KUKA KRL data list: ps_b_etb_res_c02.dat

&ACCESS RVO1
&COMMENT Solda Atego ETB
DEFDAT ps_b_etb_res_c02
;FOLD EXTERNAL DECLARATIONS;%{PE}%V2.2.2,%MKUKATPBASIS,%CEXT,%VCOMMON,%P
;FOLD BAS EXT;%{PE}%V2.2.2,%MKUKATPBASIS,%CEXT,%VEXT,%P
EXT  BAS (BAS_COMMAND  :IN,REAL  :IN )
DECL INT SUCCESS
;ENDFOLD
;FOLD A10 EXT;%{E}%V2.2.2,%MKUKATPARC,%CEXT,%VEXT,%P
EXT  A10 (A_CMD_T  :IN,A_STRT_T  :IN,A_WELD_T  :IN,A_END_T  :IN,INT  :IN )
;ENDFOLD
;FOLD A20 EXT;%{E}%V2.2.2,%MKUKATPA20,%CEXT,%VEXT,%P
EXT  A20 (INT  :IN,WELD_ST  :IN,WELD_FI  :IN,INT  :IN )
;ENDFOLD
;FOLD GRIPPER EXT;%{E}%V2.2.2,%MKUKATPGRIPPER,%CEXT,%VEXT,%P
EXT  H50 (INT  :IN,INT  :IN,INT  :IN,GRP_TYP  :IN )
;ENDFOLD
;FOLD SPOT EXT;%{E}%V2.2.2,%MKUKATPSPOT,%CEXT,%VEXT,%P
EXT  USERSPOT (S_COMMAND  :IN,SPOT_TYPE  :IN )
;ENDFOLD
;FOLD TOUCHSENSE EXT;%{E}%V2.2.2,%MKUKATPTS,%CEXT,%VEXT,%P
EXT  H70 (INT  :IN,SRCH_TYP_2  :OUT,E6POS  :IN,SRCH_TYP_3  :IN,SRCH_TYP_2  :IN,SRCH_TYP_2  :IN,SRCH_TYP_2  :IN,SRCH_TYP_2  :IN,SRCH_TYP_2  :IN,INT  :IN )
;ENDFOLD
;FOLD USER EXT;%{}%V2.2.2,%MKUKATPUSER,%CEXT,%VEXT,%P
;Make here your modifications
;ENDFOLD
;ENDFOLD

DECL FDAT Fl005={TOOL_NO 3,BASE_NO 3,IPO_FRAME #BASE}
DECL PDAT PP_OLP2={VEL 100.0,ACC 100.0,APO_DIST 0.0}
DECL E6POS Xl005={x -259.953003,y 860.291992,z 674.213013,a 106.465103,b 65.7322998,c -50.9701004,s 2,t 42}
DECL FDAT Fl010={TOOL_NO 3,BASE_NO 3,IPO_FRAME #BASE}
DECL PDAT PP_OLP3={VEL 100.0,ACC 100.0,APO_DIST 0.0}
DECL E6POS Xl010={x 238.578995,y 878.294983,z 634.81897,a 106.465103,b 65.7322998,c -50.9701004,s 2,t 43}
DECL FDAT Fl015={TOOL_NO 3,BASE_NO 3,IPO_FRAME #BASE}
DECL PDAT PP_OLP4={VEL 100.0,ACC 100.0,APO_DIST 0.0}
DECL E6POS Xl015={x 233.995102,y 927.062683,z 508.398987,a 106.4627,b 65.7314301,c -48.9741592,s 2,t 43,e1 0.0,e2 0.0,e3 0.0,e4 0.0,e5 0.0,e6 0.0}
DECL LDAT LL_OLP1={VEL 2.0,ACC 100.0,APO_DIST 0.0,APO_FAC 0.0}
DECL FDAT Fl020={TOOL_NO 3,BASE_NO 3,IPO_FRAME #BASE}
DECL PDAT PP_OLP5={VEL 100.0,ACC 100.0,APO_DIST 0.0}
DECL E6POS Xl020={x 240.050705,y 924.635925,z 506.612305,a 106.462997,b 65.7332382,c -48.9725304,s 2,t 43,e1 0.0,e2 0.0,e3 0.0,e4 0.0,e5 0.0,e6 0.0}
DECL FDAT Fl025={TOOL_NO 3,BASE_NO 3,IPO_FRAME #BASE}
DECL PDAT PP_OLP6={VEL 100.0,ACC 100.0,APO_DIST 0.0}
DECL E6POS Xl025={x 230.037399,y 926.909119,z 610.785889,a 106.4646,b 65.7323837,c -48.9705811,s 2,t 43,e1 0.0,e2 0.0,e3 0.0,e4 0.0,e5 0.0,e6 0.0}
DECL FDAT Fl030={TOOL_NO 3,BASE_NO 3,IPO_FRAME #BASE}
DECL PDAT PP_OLP7={VEL 100.0,ACC 100.0,APO_DIST 0.0}
DECL E6POS Xl030={x 193.569397,y 878.43573,z 618.731201,a 136.368896,b 76.3886337,c -42.6437798,s 2,t 43,e1 0.0,e2 0.0,e3 0.0,e4 0.0,e5 0.0,e6 0.0}
DECL E6POS Xl011={x 216.297104,y 817.987915,z 621.025818,a -90.0010071,b 86.8945236,c 89.9989166,s 2,t 43,e1 0.0,e2 0.0,e3 0.0,e4 0.0,e5 0.0,e6 0.0}
DECL FDAT Fl011={TOOL_NO 3,BASE_NO 3,IPO_FRAME #BASE}
DECL PDAT PP_OLP11={VEL 100.0,ACC 100.0,APO_DIST 0.0}
DECL E6POS Xl016={x 211.330002,y 837.989685,z 424.030212,a -89.9980164,b 86.8946533,c 90.0018005,s 2,t 43,e1 0.0,e2 0.0,e3 0.0,e4 0.0,e5 0.0,e6 0.0}
DECL FDAT Fl016={TOOL_NO 3,BASE_NO 3,IPO_FRAME #BASE}
DECL PDAT PP_OLP12={VEL 100.0,ACC 100.0,APO_DIST 0.0}
DECL E6POS XSWP_60_7354={x 203.809906,y 837.713989,z 419.105103,a -90.024231,b 86.8921432,c 89.974617,s 2,t 43,e1 0.0,e2 0.0,e3 0.0,e4 0.0,e5 0.0,e6 0.0}
DECL FDAT FSWP_60_7354={TOOL_NO 3,BASE_NO 3,IPO_FRAME #BASE}
DECL LDAT LL_OLP2={VEL 2.0,ACC 100.0,APO_DIST 0.0,APO_FAC 0.0}
DECL E6POS XSWP_60_7356={x 204.900299,y 813.062012,z 427.303589,a -90.0252304,b 86.8959122,c 89.9749298,s 2,t 43,e1 0.0,e2 0.0,e3 0.0,e4 0.0,e5 0.0,e6 0.0}
DECL FDAT FSWP_60_7356={TOOL_NO 3,BASE_NO 3,IPO_FRAME #BASE}
DECL LDAT LL_OLP3={VEL 2.0,ACC 100.0,APO_DIST 0.0,APO_FAC 0.0}
DECL E6POS XSWP_60_7358={x 205.666595,y 785.228699,z 444.857788,a -90.0419312,b 86.8953781,c 89.9582901,s 2,t 43,e1 0.0,e2 0.0,e3 0.0,e4 0.0,e5 0.0,e6 0.0}
DECL FDAT FSWP_60_7358={TOOL_NO 3,BASE_NO 3,IPO_FRAME #BASE}
DECL LDAT LL_OLP4={VEL 2.0,ACC 100.0,APO_DIST 0.0,APO_FAC 0.0}
DECL E6POS XSWP_60_7360={x 203.261703,y 756.455627,z 466.485809,a -89.9985809,b 86.8937683,c 90.0012436,s 2,t 43,e1 0.0,e2 0.0,e3 0.0,e4 0.0,e5 0.0,e6 0.0}
DECL FDAT FSWP_60_7360={TOOL_NO 3,BASE_NO 3,IPO_FRAME #BASE}
DECL LDAT LL_OLP5={VEL 2.0,ACC 100.0,APO_DIST 0.0,APO_FAC 0.0}
DECL E6POS XSWP_60_7362={x 206.944794,y 725.337585,z 475.673492,a 89.9988937,b 70.9206924,c -90.0019226,s 2,t 43,e1 0.0,e2 0.0,e3 0.0,e4 0.0,e5 0.0,e6 0.0}
DECL FDAT FSWP_60_7362={TOOL_NO 3,BASE_NO 3,IPO_FRAME #BASE}
DECL LDAT LL_OLP6={VEL 2.0,ACC 100.0,APO_DIST 0.0,APO_FAC 0.0}
DECL E6POS XSWP_60_7364={x 206.622696,y 692.928894,z 476.588287,a -90.0024414,b 86.1575623,c 89.9975586,s 2,t 43,e1 0.0,e2 0.0,e3 0.0,e4 0.0,e5 0.0,e6 0.0}
DECL FDAT FSWP_60_7364={TOOL_NO 3,BASE_NO 3,IPO_FRAME #BASE}
DECL LDAT LL_OLP7={VEL 2.0,ACC 100.0,APO_DIST 0.0,APO_FAC 0.0}
DECL E6POS XSWP_60_7366={x 203.315002,y 660.348389,z 476.359894,a -90.0006638,b 56.1120415,c 89.9992981,s 2,t 43,e1 0.0,e2 0.0,e3 0.0,e4 0.0,e5 0.0,e6 0.0}
DECL FDAT FSWP_60_7366={TOOL_NO 3,BASE_NO 3,IPO_FRAME #BASE}
DECL LDAT LL_OLP8={VEL 2.0,ACC 100.0,APO_DIST 0.0,APO_FAC 0.0}
DECL E6POS XSWP_60_7368={x 206.116501,y 634.32843,z 476.098907,a -90.0014801,b 58.2454681,c 90.0003967,s 2,t 43,e1 0.0,e2 0.0,e3 0.0,e4 0.0,e5 0.0,e6 0.0}
DECL FDAT FSWP_60_7368={TOOL_NO 3,BASE_NO 3,IPO_FRAME #BASE}
DECL LDAT LL_OLP9={VEL 2.0,ACC 100.0,APO_DIST 0.0,APO_FAC 0.0}
DECL E6POS XSWP_60_7370={x 205.649307,y 608.364075,z 476.227295,a -90.000618,b 59.0425911,c 89.9998627,s 2,t 43,e1 0.0,e2 0.0,e3 0.0,e4 0.0,e5 0.0,e6 0.0}
DECL FDAT FSWP_60_7370={TOOL_NO 3,BASE_NO 3,IPO_FRAME #BASE}
DECL LDAT LL_OLP10={VEL 2.0,ACC 100.0,APO_DIST 0.0,APO_FAC 0.0}
DECL E6POS XSWP_60_7372={x 207.227097,y 582.377502,z 476.378601,a -90.0000229,b 59.7199898,c 90.0000229,s 2,t 43,e1 0.0,e2 0.0,e3 0.0,e4 0.0,e5 0.0,e6 0.0}
DECL FDAT FSWP_60_7372={TOOL_NO 3,BASE_NO 3,IPO_FRAME #BASE}
DECL LDAT LL_OLP11={VEL 2.0,ACC 100.0,APO_DIST 0.0,APO_FAC 0.0}
DECL E6POS XSWP_60_7374={x 206.739594,y 556.385376,z 476.24881,a -89.9996872,b 60.0724792,c 89.9999695,s 2,t 43,e1 0.0,e2 0.0,e3 0.0,e4 0.0,e5 0.0,e6 0.0}
DECL FDAT FSWP_60_7374={TOOL_NO 3,BASE_NO 3,IPO_FRAME #BASE}
DECL LDAT LL_OLP12={VEL 2.0,ACC 100.0,APO_DIST 0.0,APO_FAC 0.0}
DECL E6POS Xl026={x 232.763107,y 556.379089,z 476.253387,a -89.9998627,b 59.855629,c 90.0001068,s 2,t 43,e1 0.0,e2 0.0,e3 0.0,e4 0.0,e5 0.0,e6 0.0}
DECL FDAT Fl026={TOOL_NO 3,BASE_NO 3,IPO_FRAME #BASE}
DECL PDAT PP_OLP14={VEL 100.0,ACC 100.0,APO_DIST 0.0}
DECL E6POS Xl031={x 237.137695,y 429.935913,z 476.3927,a -90.001503,b 59.8552017,c 89.9993286,s 2,t 43,e1 0.0,e2 0.0,e3 0.0,e4 0.0,e5 0.0,e6 0.0}
DECL FDAT Fl031={TOOL_NO 3,BASE_NO 3,IPO_FRAME #BASE}
DECL PDAT PP_OLP15={VEL 100.0,ACC 100.0,APO_DIST 0.0}
DECL E6POS XSWP_60_7376={x 205.848206,y 441.043304,z 482.712006,a -89.9979706,b 60.0047493,c 90.0008774,s 2,t 43,e1 0.0,e2 0.0,e3 0.0,e4 0.0,e5 0.0,e6 0.0}
DECL FDAT FSWP_60_7376={TOOL_NO 3,BASE_NO 3,IPO_FRAME #BASE}
DECL LDAT LL_OLP13={VEL 2.0,ACC 100.0,APO_DIST 0.0,APO_FAC 0.0}
DECL E6POS XSWP_60_7378={x 206.973907,y 431.014099,z 441.041809,a -89.9991226,b 61.5301018,c 90.0008698,s 2,t 43,e1 0.0,e2 0.0,e3 0.0,e4 0.0,e5 0.0,e6 0.0}
DECL FDAT FSWP_60_7378={TOOL_NO 3,BASE_NO 3,IPO_FRAME #BASE}
DECL LDAT LL_OLP14={VEL 2.0,ACC 100.0,APO_DIST 0.0,APO_FAC 0.0}
DECL E6POS XSWP_60_7380={x 206.840393,y 416.639099,z 400.304108,a -89.9998703,b 62.6937904,c 90.0006027,s 2,t 43,e1 0.0,e2 0.0,e3 0.0,e4 0.0,e5 0.0,e6 0.0}
DECL FDAT FSWP_60_7380={TOOL_NO 3,BASE_NO 3,IPO_FRAME #BASE}
DECL LDAT LL_OLP15={VEL 2.0,ACC 100.0,APO_DIST 0.0,APO_FAC 0.0}
DECL E6POS XSWP_60_7220={x 205.599396,y 39.2980804,z 386.423615,a -89.9959183,b 44.4748917,c 89.9934921,s 2,t 43,e1 0.0,e2 0.0,e3 0.0,e4 0.0,e5 0.0,e6 0.0}
DECL FDAT FSWP_60_7220={TOOL_NO 3,BASE_NO 3,IPO_FRAME #BASE}
DECL E6POS XSWP_60_7222={x 206.282593,y 88.0883484,z 386.359711,a -89.9976273,b 44.4760399,c 89.9922333,s 2,t 43,e1 0.0,e2 0.0,e3 0.0,e4 0.0,e5 0.0,e6 0.0}
DECL FDAT FSWP_60_7222={TOOL_NO 3,BASE_NO 3,IPO_FRAME #BASE}
DECL LDAT LL_OLP31={VEL 2.0,ACC 50.0,APO_DIST 0.0,APO_FAC 0.0}
DECL LDAT LL_OLP32={VEL 2.0,ACC 50.0,APO_DIST 0.0,APO_FAC 0.0}
DECL LDAT LL_OLP33={VEL 2.0,ACC 100.0,APO_DIST 0.0,APO_FAC 0.0}
DECL LDAT LL_OLP34={VEL 2.0,ACC 100.0,APO_DIST 0.0,APO_FAC 0.0}
DECL E6POS XSWP_60_7260={x 181.102097,y 50.2497406,z 492.070099,a -80.3131027,b 32.1295509,c 107.793098,s 2,t 11,e1 0.0,e2 0.0,e3 0.0,e4 0.0,e5 0.0,e6 0.0}
DECL FDAT FSWP_60_7260={TOOL_NO 3,BASE_NO 3,IPO_FRAME #BASE}
DECL E6POS XSWP_60_7261={x 180.671097,y 1.26443899,z 490.916901,a -80.5087128,b 31.6135597,c 107.6959,s 2,t 11,e1 0.0,e2 0.0,e3 0.0,e4 0.0,e5 0.0,e6 0.0}
DECL FDAT FSWP_60_7261={TOOL_NO 3,BASE_NO 3,IPO_FRAME #BASE}
DECL LDAT LL_OLP36={VEL 2.0,ACC 100.0,APO_DIST 0.0,APO_FAC 0.0}
DECL LDAT LL_OLP37={VEL 2.0,ACC 100.0,APO_DIST 0.0,APO_FAC 0.0}
DECL LDAT LL_OLP38={VEL 2.0,ACC 100.0,APO_DIST 0.0,APO_FAC 0.0}
DECL E6POS Xl086={x 160.914307,y 87.6342468,z 584.528687,a -71.1530838,b 50.3254509,c 113.916496,s 2,t 43,e1 0.0,e2 0.0,e3 0.0,e4 0.0,e5 0.0,e6 0.0}
DECL FDAT Fl086={TOOL_NO 3,BASE_NO 3,IPO_FRAME #BASE}
DECL PDAT PP_OLP49={VEL 100.0,ACC 100.0,APO_DIST 0.0}
DECL E6POS Xl091={x 172.296906,y 391.390808,z 683.738708,a -90.0011826,b 46.4089699,c 90.0007324,s 2,t 43,e1 0.0,e2 0.0,e3 0.0,e4 0.0,e5 0.0,e6 0.0}
DECL FDAT Fl091={TOOL_NO 3,BASE_NO 3,IPO_FRAME #BASE}
DECL PDAT PP_OLP50={VEL 100.0,ACC 100.0,APO_DIST 0.0}
DECL E6POS Xl096={x -352.044708,y 791.362305,z 674.194885,a 102.528297,b 65.7295227,c -50.9826317,s 2,t 42,e1 0.0,e2 0.0,e3 0.0,e4 0.0,e5 0.0,e6 0.0}
DECL FDAT Fl096={TOOL_NO 3,BASE_NO 3,IPO_FRAME #BASE}
DECL PDAT PP_OLP51={VEL 100.0,ACC 100.0,APO_DIST 0.0}
DECL E6POS XSWP_60_9320={x 233.906906,y 930.794983,z 509.773987,a 106.517899,b 65.7420273,c -48.8959618,s 2,t 43,e1 0.0,e2 0.0,e3 0.0,e4 0.0,e5 0.0,e6 0.0}
DECL FDAT FSWP_60_9320={TOOL_NO 3,BASE_NO 3,IPO_FRAME #BASE}
DECL E6POS XP6={x -1383.52795,y 1084.21204,z 300.229401,a 152.116806,b 8.17701721,c 8.23256302,s 2,t 42,e1 0.0,e2 0.0,e3 0.0,e4 0.0,e5 0.0,e6 0.0}
DECL FDAT FP6={TOOL_NO 3,BASE_NO 3,IPO_FRAME #BASE}
DECL PDAT PPDAT6={VEL 100.0,ACC 100.0,APO_DIST 0.0}
DECL E6POS XP7={x 211.5793,y 905.759277,z 610.608276,a 118.261002,b 68.8623581,c -44.6343498,s 2,t 43,e1 0.0,e2 0.0,e3 0.0,e4 0.0,e5 0.0,e6 0.0}
DECL FDAT FP7={TOOL_NO 3,BASE_NO 3,IPO_FRAME #BASE}
DECL PDAT PPDAT7={VEL 100.0,ACC 100.0,APO_DIST 0.0}
DECL SPOT_SUGG_T LAST_SPOT={GUN[] "3                       ",RETR_CMD[] "#OPN                    ",CHOISE[] "#FIRST                  ",CLO_TM[] "1                       ",PGNO1[] "197                     ",PRESS1[] "0                       ",PGNO2[] "1                       ",PRESS2[] "0                       ",SPOT_PARAMS[] "NORMAL                  "}
DECL BASIS_SUGG_T LAST_BASIS={POINT1[] "SWP_60_9234             ",POINT2[] "SWP_60_9234             ",CP_PARAMS[] "CPDAT30                 ",PTP_PARAMS[] "PDAT38                  ",CONT[] "                        ",CP_VEL[] "2                       ",PTP_VEL[] "100                     "}
DECL E6POS XSWP_60_7258={x 177.344299,y 91.2774734,z 492.510498,a -80.9878082,b 30.2983799,c 107.447899,s 2,t 11,e1 0.0,e2 0.0,e3 0.0,e4 0.0,e5 0.0,e6 0.0}
DECL FDAT FSWP_60_7258={TOOL_NO 3,BASE_NO 3,IPO_FRAME #BASE}
DECL E6POS XSWP_60_7217={x 212.0215,y -5.72816896,z 386.457611,a -89.9976273,b 44.4766617,c 89.9928436,s 2,t 43,e1 0.0,e2 0.0,e3 0.0,e4 0.0,e5 0.0,e6 0.0}
DECL FDAT FSWP_60_7217={TOOL_NO 3,BASE_NO 3,IPO_FRAME #BASE}
DECL E6POS XSWP_60_7218={x 230.446198,y 232.953796,z 499.446594,a -89.995369,b 44.4764595,c 89.9949036,s 2,t 43,e1 0.0,e2 0.0,e3 0.0,e4 0.0,e5 0.0,e6 0.0}
DECL FDAT FSWP_60_7218={TOOL_NO 3,BASE_NO 3,IPO_FRAME #BASE}
DECL PDAT PPDAT1={VEL 100.0,ACC 100.0,APO_DIST 0.0}
DECL E6POS XSWP_60_7253={x 183.271103,y -168.511398,z 488.607788,a -80.492569,b 31.5890808,c 107.705902,s 2,t 43,e1 0.0,e2 0.0,e3 0.0,e4 0.0,e5 0.0,e6 0.0}
DECL FDAT FSWP_60_7253={TOOL_NO 3,BASE_NO 3,IPO_FRAME #BASE}
DECL E6POS XSWP_60_7255={x 182.816605,y -136.932495,z 488.353302,a -80.4999466,b 31.6015491,c 107.701401,s 2,t 43,e1 0.0,e2 0.0,e3 0.0,e4 0.0,e5 0.0,e6 0.0}
DECL FDAT FSWP_60_7255={TOOL_NO 3,BASE_NO 3,IPO_FRAME #BASE}
DECL E6POS XSWP_60_7257={x 182.301605,y -88.3556519,z 488.131897,a -80.5033569,b 31.6069908,c 107.6978,s 2,t 43,e1 0.0,e2 0.0,e3 0.0,e4 0.0,e5 0.0,e6 0.0}
DECL FDAT FSWP_60_7257={TOOL_NO 3,BASE_NO 3,IPO_FRAME #BASE}
DECL E6POS XSWP_60_7262={x 180.669205,y 1.25821102,z 490.930298,a -80.508873,b 31.6130199,c 107.696198,s 2,t 11,e1 0.0,e2 0.0,e3 0.0,e4 0.0,e5 0.0,e6 0.0}
DECL FDAT FSWP_60_7262={TOOL_NO 3,BASE_NO 3,IPO_FRAME #BASE}
DECL SPOT_TYPE SNORMAL
DECL SPOT_TYPE SNORMAL28
DECL E6POS XP15={x -800.207581,y 1052.86096,z 371.426514,a 42.3493195,b -1.00002205,c -26.3774109,s 2,t 42,e1 0.0,e2 0.0,e3 0.0,e4 0.0,e5 0.0,e6 0.0}
DECL FDAT FP15={TOOL_NO 1,BASE_NO 3,IPO_FRAME #BASE}
DECL PDAT PPDAT2={VEL 100.0,ACC 100.0,APO_DIST 100.0}
DECL E6POS Xl048={x 235.096298,y 205.879898,z 399.392609,a -89.9929504,b 44.4753685,c 89.9981766,s 2,t 43,e1 0.0,e2 0.0,e3 0.0,e4 0.0,e5 0.0,e6 0.0}
DECL FDAT Fl048={TOOL_NO 3,BASE_NO 3,IPO_FRAME #BASE}
DECL PDAT PP_OLP53={VEL 100.0,ACC 100.0,APO_DIST 0.0}
DECL LDAT LL_OLP50={VEL 2.0,ACC 100.0,APO_DIST 0.0,APO_FAC 0.0}
DECL SPOT_TYPE SNORMAL29
DECL LDAT LCPDAT5={VEL 2.0,ACC 100.0,APO_DIST 100.0,APO_FAC 50.0}
DECL LDAT LCPDAT6={VEL 2.0,ACC 100.0,APO_DIST 100.0,APO_FAC 50.0}
DECL E6POS XP16={x 208.831604,y -34.5271187,z 495.562012,a -80.5012817,b 31.5980301,c 107.702202,s 2,t 11,e1 0.0,e2 0.0,e3 0.0,e4 0.0,e5 0.0,e6 0.0}
DECL FDAT FP16={TOOL_NO 3,BASE_NO 3,IPO_FRAME #BASE}
DECL LDAT LCPDAT7={VEL 2.0,ACC 50.0,APO_DIST 100.0,APO_FAC 50.0}
DECL E6POS XSWP_60_7381={x 206.840393,y 416.639099,z 400.304108,a -89.9998703,b 62.6937904,c 90.0006027,s 2,t 43,e1 0.0,e2 0.0,e3 0.0,e4 0.0,e5 0.0,e6 0.0}
DECL FDAT FSWP_60_7381={TOOL_NO 3,BASE_NO 3,IPO_FRAME #BASE}
DECL LDAT LL_OLP16={VEL 2.0,ACC 100.0,APO_DIST 0.0,APO_FAC 0.0}
DECL SPOT_TYPE SNORMAL13
DECL E6POS XSWP_60_7382={x 206.840393,y 416.639099,z 400.304108,a -89.9998703,b 62.6937904,c 90.0006027,s 2,t 43,e1 0.0,e2 0.0,e3 0.0,e4 0.0,e5 0.0,e6 0.0}
DECL FDAT FSWP_60_7382={TOOL_NO 3,BASE_NO 3,IPO_FRAME #BASE}
DECL LDAT LL_OLP17={VEL 2.0,ACC 100.0,APO_DIST 0.0,APO_FAC 0.0}
DECL E6POS XSWP_60_7383={x 206.840393,y 416.639099,z 400.304108,a -89.9998703,b 62.6937904,c 90.0006027,s 2,t 43,e1 0.0,e2 0.0,e3 0.0,e4 0.0,e5 0.0,e6 0.0}
DECL FDAT FSWP_60_7383={TOOL_NO 3,BASE_NO 3,IPO_FRAME #BASE}
DECL LDAT LL_OLP18={VEL 2.0,ACC 100.0,APO_DIST 0.0,APO_FAC 0.0}
DECL E6POS XSWP_60_7384={x 206.840393,y 416.639099,z 400.304108,a -89.9998703,b 62.6937904,c 90.0006027,s 2,t 43,e1 0.0,e2 0.0,e3 0.0,e4 0.0,e5 0.0,e6 0.0}
DECL FDAT FSWP_60_7384={TOOL_NO 3,BASE_NO 3,IPO_FRAME #BASE}
DECL LDAT LL_OLP19={VEL 2.0,ACC 100.0,APO_DIST 0.0,APO_FAC 0.0}
DECL E6POS XSWP_60_7385={x 206.840393,y 416.639099,z 400.304108,a -89.9998703,b 62.6937904,c 90.0006027,s 2,t 43,e1 0.0,e2 0.0,e3 0.0,e4 0.0,e5 0.0,e6 0.0}
DECL FDAT FSWP_60_7385={TOOL_NO 3,BASE_NO 3,IPO_FRAME #BASE}
DECL LDAT LL_OLP20={VEL 2.0,ACC 100.0,APO_DIST 0.0,APO_FAC 0.0}
DECL E6POS XP17={x 487.528015,y 470.183289,z 402.488708,a 89.9994965,b -2.90493488,c -90.0005722,s 2,t 43,e1 0.0,e2 0.0,e3 0.0,e4 0.0,e5 0.0,e6 0.0}
DECL FDAT FP17={TOOL_NO 1,BASE_NO 3,IPO_FRAME #BASE}
DECL PDAT PPDAT5={VEL 100.0,ACC 80.0,APO_DIST 100.0}
DECL E6POS XSWP_60_9230={x 213.558807,y 372.876587,z 385.620087,a -89.9933701,b 62.6980019,c 90.0031433,s 2,t 43,e1 0.0,e2 0.0,e3 0.0,e4 0.0,e5 0.0,e6 0.0}
DECL FDAT FSWP_60_9230={TOOL_NO 3,BASE_NO 3,IPO_FRAME #BASE}
DECL E6POS XSWP_60_7230={x 206.551697,y 281.323212,z 384.273712,a -89.9992828,b 62.6938591,c 90.0016403,s 2,t 43,e1 0.0,e2 0.0,e3 0.0,e4 0.0,e5 0.0,e6 0.0}
DECL FDAT FSWP_60_7230={TOOL_NO 3,BASE_NO 3,IPO_FRAME #BASE}
DECL E6POS XSWP_60_9224={x 212.6707,y 237.668198,z 383.0448,a -90.0036316,b 62.6945114,c 89.9956436,s 2,t 43,e1 0.0,e2 0.0,e3 0.0,e4 0.0,e5 0.0,e6 0.0}
DECL FDAT FSWP_60_9224={TOOL_NO 3,BASE_NO 3,IPO_FRAME #BASE}
DECL E6POS XSWP_60_9222={x 213.009705,y 187.713104,z 381.806488,a -90.0050735,b 62.6927795,c 89.9951172,s 2,t 43,e1 0.0,e2 0.0,e3 0.0,e4 0.0,e5 0.0,e6 0.0}
DECL FDAT FSWP_60_9222={TOOL_NO 3,BASE_NO 3,IPO_FRAME #BASE}
DECL E6POS XSWP_60_9220={x 212.403503,y 141.233597,z 380.69751,a -90.0037689,b 54.2511902,c 89.9956436,s 2,t 43,e1 0.0,e2 0.0,e3 0.0,e4 0.0,e5 0.0,e6 0.0}
DECL FDAT FSWP_60_9220={TOOL_NO 3,BASE_NO 3,IPO_FRAME #BASE}
DECL E6POS XP18={x 479.408508,y 208.821899,z 388.631012,a 90.0012131,b -2.90534997,c -90.0033875,s 2,t 43,e1 0.0,e2 0.0,e3 0.0,e4 0.0,e5 0.0,e6 0.0}
DECL FDAT FP18={TOOL_NO 1,BASE_NO 3,IPO_FRAME #BASE}
DECL PDAT PPDAT8={VEL 100.0,ACC 80.0,APO_DIST 100.0}
DECL E6POS XSWP_60_7223={x 211.064697,y 88.1381378,z 386.404205,a -89.9957275,b 44.4758797,c 89.9949112,s 2,t 43,e1 0.0,e2 0.0,e3 0.0,e4 0.0,e5 0.0,e6 0.0}
DECL FDAT FSWP_60_7223={TOOL_NO 3,BASE_NO 3,IPO_FRAME #BASE}
DECL LDAT LCPDAT8={VEL 2.0,ACC 100.0,APO_DIST 100.0,APO_FAC 50.0}
DECL SPOT_TYPE SNORMAL1
DECL E6POS XSWP_60_7219={x 212.021896,y -5.72421885,z 386.506012,a -89.9952469,b 44.4766808,c 89.9958267,s 2,t 43,e1 0.0,e2 0.0,e3 0.0,e4 0.0,e5 0.0,e6 0.0}
DECL FDAT FSWP_60_7219={TOOL_NO 3,BASE_NO 3,IPO_FRAME #BASE}
DECL LDAT LL_OLP51={VEL 2.0,ACC 100.0,APO_DIST 0.0,APO_FAC 0.0}
DECL E6POS XP19={x 456.774689,y 152.085098,z 534.078979,a 82.0662766,b 27.2542496,c -106.930702,s 2,t 11,e1 0.0,e2 0.0,e3 0.0,e4 0.0,e5 0.0,e6 0.0}
DECL FDAT FP19={TOOL_NO 1,BASE_NO 3,IPO_FRAME #BASE}
DECL PDAT PPDAT9={VEL 100.0,ACC 80.0,APO_DIST 100.0}
DECL E6POS XP20={x 463.799011,y 181.4142,z 472.935089,a 88.6661911,b 4.65849304,c -105.848,s 2,t 43,e1 0.0,e2 0.0,e3 0.0,e4 0.0,e5 0.0,e6 0.0}
DECL FDAT FP20={TOOL_NO 1,BASE_NO 3,IPO_FRAME #BASE}
DECL PDAT PPDAT10={VEL 100.0,ACC 80.0,APO_DIST 100.0}
DECL E6POS XSWP_60_7259={x 186.947998,y 91.3792191,z 492.51651,a -80.987381,b 30.2990799,c 107.448097,s 2,t 11,e1 0.0,e2 0.0,e3 0.0,e4 0.0,e5 0.0,e6 0.0}
DECL FDAT FSWP_60_7259={TOOL_NO 3,BASE_NO 3,IPO_FRAME #BASE}
DECL LDAT LL_OLP39={VEL 2.0,ACC 100.0,APO_DIST 0.0,APO_FAC 0.0}
DECL SPOT_TYPE SNORMAL36
DECL E6POS XSWP_60_7263={x 186.947998,y 91.3792191,z 492.51651,a -80.987381,b 30.2990799,c 107.448097,s 2,t 11,e1 0.0,e2 0.0,e3 0.0,e4 0.0,e5 0.0,e6 0.0}
DECL FDAT FSWP_60_7263={TOOL_NO 3,BASE_NO 3,IPO_FRAME #BASE}
DECL LDAT LL_OLP40={VEL 2.0,ACC 100.0,APO_DIST 0.0,APO_FAC 0.0}
DECL E6POS XSWP_60_7264={x 186.947998,y 91.3792191,z 492.51651,a -80.987381,b 30.2990799,c 107.448097,s 2,t 11,e1 0.0,e2 0.0,e3 0.0,e4 0.0,e5 0.0,e6 0.0}
DECL FDAT FSWP_60_7264={TOOL_NO 3,BASE_NO 3,IPO_FRAME #BASE}
DECL LDAT LL_OLP41={VEL 2.0,ACC 100.0,APO_DIST 0.0,APO_FAC 0.0}
DECL E6POS XSWP_60_7265={x 186.947998,y 91.3792191,z 492.51651,a -80.987381,b 30.2990799,c 107.448097,s 2,t 11,e1 0.0,e2 0.0,e3 0.0,e4 0.0,e5 0.0,e6 0.0}
DECL FDAT FSWP_60_7265={TOOL_NO 3,BASE_NO 3,IPO_FRAME #BASE}
DECL LDAT LL_OLP42={VEL 2.0,ACC 100.0,APO_DIST 0.0,APO_FAC 0.0}
DECL E6POS XSWP_60_7266={x 186.947998,y 91.3792191,z 492.51651,a -80.987381,b 30.2990799,c 107.448097,s 2,t 11,e1 0.0,e2 0.0,e3 0.0,e4 0.0,e5 0.0,e6 0.0}
DECL FDAT FSWP_60_7266={TOOL_NO 3,BASE_NO 3,IPO_FRAME #BASE}
DECL LDAT LL_OLP43={VEL 2.0,ACC 100.0,APO_DIST 0.0,APO_FAC 0.0}
DECL E6POS XSWP_60_7267={x 186.947998,y 91.3792191,z 492.51651,a -80.987381,b 30.2990799,c 107.448097,s 2,t 11,e1 0.0,e2 0.0,e3 0.0,e4 0.0,e5 0.0,e6 0.0}
DECL FDAT FSWP_60_7267={TOOL_NO 3,BASE_NO 3,IPO_FRAME #BASE}
DECL LDAT LL_OLP44={VEL 2.0,ACC 100.0,APO_DIST 0.0,APO_FAC 0.0}
DECL E6POS XSWP_60_7268={x 186.947998,y 91.3792191,z 492.51651,a -80.987381,b 30.2990799,c 107.448097,s 2,t 11,e1 0.0,e2 0.0,e3 0.0,e4 0.0,e5 0.0,e6 0.0}
DECL FDAT FSWP_60_7268={TOOL_NO 3,BASE_NO 3,IPO_FRAME #BASE}
DECL LDAT LL_OLP45={VEL 2.0,ACC 100.0,APO_DIST 0.0,APO_FAC 0.0}
DECL E6POS XSWP_60_7269={x 186.947998,y 91.3792191,z 492.51651,a -80.987381,b 30.2990799,c 107.448097,s 2,t 11,e1 0.0,e2 0.0,e3 0.0,e4 0.0,e5 0.0,e6 0.0}
DECL FDAT FSWP_60_7269={TOOL_NO 3,BASE_NO 3,IPO_FRAME #BASE}
DECL LDAT LL_OLP46={VEL 2.0,ACC 100.0,APO_DIST 0.0,APO_FAC 0.0}
DECL E6POS XSWP_60_7270={x 186.947998,y 91.3792191,z 492.51651,a -80.987381,b 30.2990799,c 107.448097,s 2,t 11,e1 0.0,e2 0.0,e3 0.0,e4 0.0,e5 0.0,e6 0.0}
DECL FDAT FSWP_60_7270={TOOL_NO 3,BASE_NO 3,IPO_FRAME #BASE}
DECL LDAT LL_OLP47={VEL 2.0,ACC 100.0,APO_DIST 0.0,APO_FAC 0.0}
DECL E6POS XSWP_60_7271={x 186.947998,y 91.3792191,z 492.51651,a -80.987381,b 30.2990799,c 107.448097,s 2,t 11,e1 0.0,e2 0.0,e3 0.0,e4 0.0,e5 0.0,e6 0.0}
DECL FDAT FSWP_60_7271={TOOL_NO 3,BASE_NO 3,IPO_FRAME #BASE}
DECL LDAT LL_OLP48={VEL 2.0,ACC 100.0,APO_DIST 0.0,APO_FAC 0.0}
DECL E6POS XSWP_60_7272={x 186.947998,y 91.3792191,z 492.51651,a -80.987381,b 30.2990799,c 107.448097,s 2,t 11,e1 0.0,e2 0.0,e3 0.0,e4 0.0,e5 0.0,e6 0.0}
DECL FDAT FSWP_60_7272={TOOL_NO 3,BASE_NO 3,IPO_FRAME #BASE}
DECL LDAT LL_OLP49={VEL 2.0,ACC 100.0,APO_DIST 0.0,APO_FAC 0.0}
DECL E6POS XSWP_60_7273={x 186.947998,y 91.3792191,z 492.51651,a -80.987381,b 30.2990799,c 107.448097,s 2,t 11,e1 0.0,e2 0.0,e3 0.0,e4 0.0,e5 0.0,e6 0.0}
DECL FDAT FSWP_60_7273={TOOL_NO 3,BASE_NO 3,IPO_FRAME #BASE}
DECL LDAT LL_OLP52={VEL 2.0,ACC 100.0,APO_DIST 0.0,APO_FAC 0.0}
DECL E6POS XSWP_60_9308={x 209.725403,y 113.234398,z 405.451508,a -73.5277405,b 45.4200516,c 112.484398,s 2,t 43,e1 0.0,e2 0.0,e3 0.0,e4 0.0,e5 0.0,e6 0.0}
DECL FDAT FSWP_60_9308={TOOL_NO 3,BASE_NO 3,IPO_FRAME #BASE}
DECL E6POS XSWP_60_9310={x 202.714798,y 113.227203,z 431.928802,a -73.5278625,b 45.4177208,c 112.4842,s 2,t 43,e1 0.0,e2 0.0,e3 0.0,e4 0.0,e5 0.0,e6 0.0}
DECL FDAT FSWP_60_9310={TOOL_NO 3,BASE_NO 3,IPO_FRAME #BASE}
DECL E6POS XSWP_60_9212={x 193.037201,y 112.178398,z 461.130707,a -73.5264206,b 45.4157715,c 112.485703,s 2,t 43,e1 0.0,e2 0.0,e3 0.0,e4 0.0,e5 0.0,e6 0.0}
DECL FDAT FSWP_60_9212={TOOL_NO 3,BASE_NO 3,IPO_FRAME #BASE}
DECL E6POS XSWP_60_9250={x 186.693405,y 130.9664,z 489.893188,a -73.5289917,b 45.4151688,c 112.485397,s 2,t 43,e1 0.0,e2 0.0,e3 0.0,e4 0.0,e5 0.0,e6 0.0}
DECL FDAT FSWP_60_9250={TOOL_NO 3,BASE_NO 3,IPO_FRAME #BASE}
DECL E6POS XSWP_60_9248={x 185.993896,y 168.512497,z 487.767792,a -73.5274277,b 45.4177895,c 112.484901,s 2,t 43,e1 0.0,e2 0.0,e3 0.0,e4 0.0,e5 0.0,e6 0.0}
DECL FDAT FSWP_60_9248={TOOL_NO 3,BASE_NO 3,IPO_FRAME #BASE}
DECL E6POS XSWP_60_9246={x 185.623703,y 206.966705,z 487.521515,a -73.5305328,b 45.4201317,c 112.481903,s 2,t 11,e1 0.0,e2 0.0,e3 0.0,e4 0.0,e5 0.0,e6 0.0}
DECL FDAT FSWP_60_9246={TOOL_NO 3,BASE_NO 3,IPO_FRAME #BASE}
DECL E6POS XSWP_60_9244={x 185.348495,y 249.794601,z 487.258301,a -73.5230865,b 45.4160995,c 112.489601,s 2,t 11,e1 0.0,e2 0.0,e3 0.0,e4 0.0,e5 0.0,e6 0.0}
DECL FDAT FSWP_60_9244={TOOL_NO 3,BASE_NO 3,IPO_FRAME #BASE}
DECL E6POS XSWP_60_9242={x 186.126694,y 285.525604,z 486.265991,a -73.5298462,b 45.417881,c 112.484497,s 2,t 11,e1 0.0,e2 0.0,e3 0.0,e4 0.0,e5 0.0,e6 0.0}
DECL FDAT FSWP_60_9242={TOOL_NO 3,BASE_NO 3,IPO_FRAME #BASE}
DECL E6POS XSWP_60_9240={x 186.675507,y 324.021393,z 486.789307,a -73.5264206,b 45.4193916,c 112.485397,s 2,t 11,e1 0.0,e2 0.0,e3 0.0,e4 0.0,e5 0.0,e6 0.0}
DECL FDAT FSWP_60_9240={TOOL_NO 3,BASE_NO 3,IPO_FRAME #BASE}
DECL E6POS XSWP_60_9238={x 185.553406,y 365.805603,z 485.38739,a -73.527153,b 45.4207191,c 112.485397,s 2,t 11,e1 0.0,e2 0.0,e3 0.0,e4 0.0,e5 0.0,e6 0.0}
DECL FDAT FSWP_60_9238={TOOL_NO 3,BASE_NO 3,IPO_FRAME #BASE}
DECL E6POS XSWP_60_9236={x 193.935104,y 386.462189,z 462.237396,a -43.1882019,b 69.0691833,c 138.712296,s 2,t 43,e1 0.0,e2 0.0,e3 0.0,e4 0.0,e5 0.0,e6 0.0}
DECL FDAT FSWP_60_9236={TOOL_NO 3,BASE_NO 3,IPO_FRAME #BASE}
DECL E6POS XSWP_60_9232={x 212.135696,y 290.268311,z 382.979889,a -90.0033493,b 62.6944618,c 89.9960098,s 2,t 43,e1 0.0,e2 0.0,e3 0.0,e4 0.0,e5 0.0,e6 0.0}
DECL FDAT FSWP_60_9232={TOOL_NO 3,BASE_NO 3,IPO_FRAME #BASE}
DECL E6POS XP21={x 433.752899,y 464.826813,z 652.343994,a 88.1901703,b 6.72100019,c -105.1064,s 2,t 11,e1 0.0,e2 0.0,e3 0.0,e4 0.0,e5 0.0,e6 0.0}
DECL FDAT FP21={TOOL_NO 1,BASE_NO 3,IPO_FRAME #BASE}
DECL PDAT PPDAT11={VEL 100.0,ACC 80.0,APO_DIST 100.0}
DECL E6POS XP22={x 442.094513,y 443.860596,z 605.23938,a 89.9556885,b -0.390171498,c -102.807098,s 2,t 43,e1 0.0,e2 0.0,e3 0.0,e4 0.0,e5 0.0,e6 0.0}
DECL FDAT FP22={TOOL_NO 1,BASE_NO 3,IPO_FRAME #BASE}
DECL PDAT PPDAT12={VEL 100.0,ACC 80.0,APO_DIST 100.0}
DECL E6POS XP23={x 458.427704,y 448.019989,z 544.208008,a 94.4578781,b -15.4476404,c -106.168999,s 2,t 43,e1 0.0,e2 0.0,e3 0.0,e4 0.0,e5 0.0,e6 0.0}
DECL FDAT FP23={TOOL_NO 1,BASE_NO 3,IPO_FRAME #BASE}
DECL PDAT PPDAT13={VEL 100.0,ACC 80.0,APO_DIST 100.0}
DECL PDAT PPDAT14={VEL 100.0,ACC 80.0,APO_DIST 100.0}
DECL LDAT LCPDAT9={VEL 2.0,ACC 100.0,APO_DIST 100.0,APO_FAC 50.0}
DECL PDAT PPDAT15={VEL 100.0,ACC 80.0,APO_DIST 100.0}
DECL LDAT LCPDAT10={VEL 2.0,ACC 100.0,APO_DIST 100.0,APO_FAC 50.0}
DECL E6POS XP12={x 468.767487,y -1397.66797,z 1152.35498,a 140.2052,b 16.2280006,c 9.75706577,s 2,t 34,e1 0.0,e2 0.0,e3 0.0,e4 0.0,e5 0.0,e6 0.0}
DECL FDAT FP12={TOOL_NO 3,BASE_NO 0,IPO_FRAME #BASE}
DECL PDAT PPDAT16={VEL 100.0,ACC 80.0,APO_DIST 100.0}
DECL E6POS XP13={x 468.767487,y -1397.66797,z 1152.35498,a 140.2052,b 16.2280006,c 9.75706577,s 2,t 34,e1 0.0,e2 0.0,e3 0.0,e4 0.0,e5 0.0,e6 0.0}
DECL FDAT FP13={TOOL_NO 3,BASE_NO 0,IPO_FRAME #BASE}
DECL PDAT PPDAT17={VEL 100.0,ACC 80.0,APO_DIST 100.0}
DECL E6POS XP14={x 468.767487,y -1397.66797,z 1152.35498,a 140.2052,b 16.2280006,c 9.75706577,s 2,t 34,e1 0.0,e2 0.0,e3 0.0,e4 0.0,e5 0.0,e6 0.0}
DECL FDAT FP14={TOOL_NO 3,BASE_NO 0,IPO_FRAME #BASE}
DECL PDAT PPDAT18={VEL 100.0,ACC 80.0,APO_DIST 100.0}
DECL E6POS XP24={x 468.767487,y -1397.66797,z 1152.35498,a 140.2052,b 16.2280006,c 9.75706577,s 2,t 34,e1 0.0,e2 0.0,e3 0.0,e4 0.0,e5 0.0,e6 0.0}
DECL FDAT FP24={TOOL_NO 3,BASE_NO 0,IPO_FRAME #BASE}
DECL PDAT PPDAT19={VEL 100.0,ACC 80.0,APO_DIST 100.0}
DECL E6POS XP25={x -384.03299,y 419.546387,z 316.5065,a 66.1975403,b -17.4831791,c -68.3892136,s 2,t 42,e1 0.0,e2 0.0,e3 0.0,e4 0.0,e5 0.0,e6 0.0}
DECL FDAT FP25={TOOL_NO 3,BASE_NO 3,IPO_FRAME #BASE}
DECL PDAT PPDAT20={VEL 100.0,ACC 80.0,APO_DIST 100.0}
DECL E6POS XP26={x 202.700699,y 221.683807,z 190.377502,a 83.5018692,b -22.9824409,c -74.4219131,s 2,t 43,e1 0.0,e2 0.0,e3 0.0,e4 0.0,e5 0.0,e6 0.0}
DECL FDAT FP26={TOOL_NO 3,BASE_NO 3,IPO_FRAME #BASE}
DECL PDAT PPDAT21={VEL 100.0,ACC 80.0,APO_DIST 100.0}
DECL E6POS XP27={x 187.651306,y 27.2828407,z 289.910187,a 88.4408417,b -40.7095108,c -87.5350037,s 2,t 43,e1 0.0,e2 0.0,e3 0.0,e4 0.0,e5 0.0,e6 0.0}
DECL FDAT FP27={TOOL_NO 3,BASE_NO 3,IPO_FRAME #BASE}
DECL LDAT LCPDAT11={VEL 2.0,ACC 100.0,APO_DIST 100.0,APO_FAC 50.0}
DECL E6POS XP28={x 186.2314,y 169.758194,z 261.008087,a 88.6298065,b -33.4667816,c -87.8612366,s 2,t 43,e1 0.0,e2 0.0,e3 0.0,e4 0.0,e5 0.0,e6 0.0}
DECL FDAT FP28={TOOL_NO 3,BASE_NO 3,IPO_FRAME #BASE}
DECL PDAT PPDAT22={VEL 100.0,ACC 80.0,APO_DIST 100.0}
DECL E6POS XSWP_60_7160={x 187.652405,y 27.2816505,z 289.94101,a 88.4419098,b -40.7085609,c -87.5364304,s 2,t 43,e1 0.0,e2 0.0,e3 0.0,e4 0.0,e5 0.0,e6 0.0}
DECL FDAT FSWP_60_7160={TOOL_NO 3,BASE_NO 3,IPO_FRAME #BASE}
DECL E6POS XP29={x 187.294296,y 62.0672302,z 289.905487,a 88.4418106,b -40.7092781,c -87.536438,s 2,t 43,e1 0.0,e2 0.0,e3 0.0,e4 0.0,e5 0.0,e6 0.0}
DECL FDAT FP29={TOOL_NO 3,BASE_NO 3,IPO_FRAME #BASE}
DECL LDAT LCPDAT12={VEL 2.0,ACC 100.0,APO_DIST 100.0,APO_FAC 50.0}
DECL E6POS XP30={x 186.636307,y 125.065102,z 289.793213,a 88.440773,b -40.712059,c -87.5349197,s 2,t 43,e1 0.0,e2 0.0,e3 0.0,e4 0.0,e5 0.0,e6 0.0}
DECL FDAT FP30={TOOL_NO 3,BASE_NO 3,IPO_FRAME #BASE}
DECL LDAT LCPDAT13={VEL 2.0,ACC 100.0,APO_DIST 100.0,APO_FAC 50.0}
DECL E6POS XSWP_60_7158={x 187.294296,y 62.0672302,z 289.905487,a 88.4418106,b -40.7092781,c -87.536438,s 2,t 43,e1 0.0,e2 0.0,e3 0.0,e4 0.0,e5 0.0,e6 0.0}
DECL FDAT FSWP_60_7158={TOOL_NO 3,BASE_NO 3,IPO_FRAME #BASE}
DECL E6POS XSWP_60_7154={x 186.636307,y 125.065102,z 289.793213,a 88.440773,b -40.712059,c -87.5349197,s 2,t 43,e1 0.0,e2 0.0,e3 0.0,e4 0.0,e5 0.0,e6 0.0}
DECL FDAT FSWP_60_7154={TOOL_NO 3,BASE_NO 3,IPO_FRAME #BASE}
DECL E6POS XSWP_60_7152={x 186.402603,y 149.349899,z 289.780396,a 88.4422379,b -40.7125282,c -87.5355225,s 2,t 43,e1 0.0,e2 0.0,e3 0.0,e4 0.0,e5 0.0,e6 0.0}
DECL FDAT FSWP_60_7152={TOOL_NO 3,BASE_NO 3,IPO_FRAME #BASE}
DECL LDAT LCPDAT14={VEL 2.0,ACC 100.0,APO_DIST 100.0,APO_FAC 50.0}
DECL E6POS XSWP_60_7150={x 184.194901,y 177.324402,z 291.644012,a 88.4415131,b -40.7133217,c -87.5351028,s 2,t 43,e1 0.0,e2 0.0,e3 0.0,e4 0.0,e5 0.0,e6 0.0}
DECL FDAT FSWP_60_7150={TOOL_NO 3,BASE_NO 3,IPO_FRAME #BASE}
DECL LDAT LCPDAT15={VEL 2.0,ACC 100.0,APO_DIST 100.0,APO_FAC 50.0}
DECL E6POS XSWP_60_7148={x 183.885406,y 206.6828,z 291.57309,a 88.4399872,b -40.71521,c -87.5329819,s 2,t 43,e1 0.0,e2 0.0,e3 0.0,e4 0.0,e5 0.0,e6 0.0}
DECL FDAT FSWP_60_7148={TOOL_NO 3,BASE_NO 3,IPO_FRAME #BASE}
DECL LDAT LCPDAT16={VEL 2.0,ACC 100.0,APO_DIST 100.0,APO_FAC 50.0}
DECL E6POS XSWP_60_7146={x 183.580994,y 235.289093,z 291.526611,a 88.4393768,b -40.7172585,c -87.5320663,s 2,t 43,e1 0.0,e2 0.0,e3 0.0,e4 0.0,e5 0.0,e6 0.0}
DECL FDAT FSWP_60_7146={TOOL_NO 3,BASE_NO 3,IPO_FRAME #BASE}
DECL LDAT LCPDAT17={VEL 2.0,ACC 100.0,APO_DIST 100.0,APO_FAC 50.0}
DECL E6POS XSWP_60_7144={x 183.271698,y 265.554901,z 291.498596,a 88.4393463,b -40.7176704,c -87.5321884,s 2,t 43,e1 0.0,e2 0.0,e3 0.0,e4 0.0,e5 0.0,e6 0.0}
DECL FDAT FSWP_60_7144={TOOL_NO 3,BASE_NO 3,IPO_FRAME #BASE}
DECL LDAT LCPDAT18={VEL 2.0,ACC 100.0,APO_DIST 100.0,APO_FAC 50.0}
DECL E6POS XSWP_60_7142={x 182.987595,y 294.084503,z 291.476715,a 88.4403076,b -40.719059,c -87.5332031,s 2,t 43,e1 0.0,e2 0.0,e3 0.0,e4 0.0,e5 0.0,e6 0.0}
DECL FDAT FSWP_60_7142={TOOL_NO 3,BASE_NO 3,IPO_FRAME #BASE}
DECL LDAT LCPDAT19={VEL 2.0,ACC 100.0,APO_DIST 100.0,APO_FAC 50.0}
DECL E6POS XSWP_60_7140={x 182.677307,y 324.696899,z 291.416504,a 88.4400635,b -40.7207718,c -87.5320663,s 2,t 43,e1 0.0,e2 0.0,e3 0.0,e4 0.0,e5 0.0,e6 0.0}
DECL FDAT FSWP_60_7140={TOOL_NO 3,BASE_NO 3,IPO_FRAME #BASE}
DECL LDAT LCPDAT20={VEL 2.0,ACC 100.0,APO_DIST 100.0,APO_FAC 50.0}
DECL E6POS XSWP_60_7136={x 183.638,y 354.853912,z 283.04599,a 88.4401169,b -40.7217407,c -87.5323563,s 2,t 43,e1 0.0,e2 0.0,e3 0.0,e4 0.0,e5 0.0,e6 0.0}
DECL FDAT FSWP_60_7136={TOOL_NO 3,BASE_NO 3,IPO_FRAME #BASE}
DECL LDAT LCPDAT21={VEL 2.0,ACC 100.0,APO_DIST 100.0,APO_FAC 50.0}
DECL E6POS XSWP_60_7137={x 188.785202,y 354.862701,z 240.309402,a 88.4393768,b -40.723999,c -87.5315781,s 2,t 43,e1 0.0,e2 0.0,e3 0.0,e4 0.0,e5 0.0,e6 0.0}
DECL FDAT FSWP_60_7137={TOOL_NO 3,BASE_NO 3,IPO_FRAME #BASE}
DECL PDAT PPDAT23={VEL 100.0,ACC 80.0,APO_DIST 100.0}
DECL E6POS XPS_30={x 8.17374325,y 352.267487,z 239.812698,a 88.4372711,b -40.7192917,c -87.5370407,s 2,t 43,e1 0.0,e2 0.0,e3 0.0,e4 0.0,e5 0.0,e6 0.0}
DECL FDAT FPS_30={TOOL_NO 3,BASE_NO 3,IPO_FRAME #BASE}
DECL PDAT PPDAT24={VEL 100.0,ACC 80.0,APO_DIST 100.0}
DECL E6POS XPS_31={x 8.17374325,y 352.267487,z 239.812698,a 88.4372711,b -40.7192917,c -87.5370407,s 2,t 43,e1 0.0,e2 0.0,e3 0.0,e4 0.0,e5 0.0,e6 0.0}
DECL FDAT FPS_31={TOOL_NO 3,BASE_NO 3,IPO_FRAME #BASE}
DECL PDAT PPDAT25={VEL 100.0,ACC 80.0,APO_DIST 100.0}
DECL E6POS XPS_32={x -352.048706,y 791.363525,z 674.182678,a 102.5298,b 65.7294617,c -50.9808998,s 2,t 42,e1 0.0,e2 0.0,e3 0.0,e4 0.0,e5 0.0,e6 0.0}
DECL FDAT FPS_32={TOOL_NO 3,BASE_NO 3,IPO_FRAME #BASE}
DECL PDAT PPDAT26={VEL 100.0,ACC 80.0,APO_DIST 100.0}
DECL E6POS XPS_33={x 187.030197,y 354.844299,z 237.620605,a 88.438652,b -40.7234612,c -87.5300064,s 2,t 43,e1 0.0,e2 0.0,e3 0.0,e4 0.0,e5 0.0,e6 0.0}
DECL FDAT FPS_33={TOOL_NO 3,BASE_NO 3,IPO_FRAME #BASE}
DECL PDAT PPDAT27={VEL 100.0,ACC 80.0,APO_DIST 100.0}
DECL E6POS XPS_34={x -938.618225,y 703.747803,z 612.635803,a 165.016998,b 23.1207695,c 13.1032801,s 2,t 42,e1 0.0,e2 0.0,e3 0.0,e4 0.0,e5 0.0,e6 0.0}
DECL FDAT FPS_34={TOOL_NO 3,BASE_NO 3,IPO_FRAME #BASE}
DECL PDAT PPDAT28={VEL 100.0,ACC 80.0,APO_DIST 100.0}
DECL E6POS XPS_35={x -373.168396,y 990.912476,z -71.8266068,a 96.466713,b 6.40488195,c -88.1943283,s 2,t 42,e1 0.0,e2 0.0,e3 0.0,e4 0.0,e5 0.0,e6 0.0}
DECL FDAT FPS_35={TOOL_NO 3,BASE_NO 3,IPO_FRAME #BASE}
DECL PDAT PPDAT29={VEL 100.0,ACC 80.0,APO_DIST 100.0}
DECL E6POS XPS_36={x -367.697113,y 444.486786,z -71.2692413,a 96.4659195,b 6.40667391,c -88.1916122,s 2,t 42,e1 0.0,e2 0.0,e3 0.0,e4 0.0,e5 0.0,e6 0.0}
DECL FDAT FPS_36={TOOL_NO 3,BASE_NO 3,IPO_FRAME #BASE}
DECL PDAT PPDAT30={VEL 100.0,ACC 80.0,APO_DIST 100.0}
DECL E6POS XPS_37={x 190.027893,y 229.223999,z 5.26974916,a 81.5058365,b -2.0061059,c -93.3127136,s 2,t 43,e1 0.0,e2 0.0,e3 0.0,e4 0.0,e5 0.0,e6 0.0}
DECL FDAT FPS_37={TOOL_NO 3,BASE_NO 3,IPO_FRAME #BASE}
DECL PDAT PPDAT31={VEL 100.0,ACC 80.0,APO_DIST 100.0}
DECL E6POS XPS_38={x 224.422607,y 239.474503,z -38.9988289,a 81.3575516,b 2.56497407,c -89.2551422,s 2,t 43,e1 0.0,e2 0.0,e3 0.0,e4 0.0,e5 0.0,e6 0.0}
DECL FDAT FPS_38={TOOL_NO 3,BASE_NO 3,IPO_FRAME #BASE}
DECL PDAT PPDAT32={VEL 100.0,ACC 80.0,APO_DIST 100.0}
DECL E6POS XSWP_60_7106={x 184.699097,y 237.990799,z -41.7804298,a 87.6008224,b 2.26465797,c -93.2121964,s 2,t 43,e1 0.0,e2 0.0,e3 0.0,e4 0.0,e5 0.0,e6 0.0}
DECL FDAT FSWP_60_7106={TOOL_NO 3,BASE_NO 3,IPO_FRAME #BASE}
DECL LDAT LCPDAT22={VEL 2.0,ACC 100.0,APO_DIST 100.0,APO_FAC 50.0}
DECL E6POS XSWP_60_7108={x 186.512299,y 265.218414,z -30.1667404,a 87.5995026,b 2.266505,c -93.2119522,s 2,t 43,e1 0.0,e2 0.0,e3 0.0,e4 0.0,e5 0.0,e6 0.0}
DECL FDAT FSWP_60_7108={TOOL_NO 3,BASE_NO 3,IPO_FRAME #BASE}
DECL LDAT LCPDAT23={VEL 2.0,ACC 100.0,APO_DIST 100.0,APO_FAC 50.0}
DECL E6POS XSWP_60_7110={x 186.609299,y 297.004791,z -18.5294304,a 87.5961838,b 2.26368904,c -93.2132187,s 2,t 43,e1 0.0,e2 0.0,e3 0.0,e4 0.0,e5 0.0,e6 0.0}
DECL FDAT FSWP_60_7110={TOOL_NO 3,BASE_NO 3,IPO_FRAME #BASE}
DECL LDAT LCPDAT24={VEL 2.0,ACC 100.0,APO_DIST 100.0,APO_FAC 50.0}
DECL E6POS XSWP_60_7112={x 182.128601,y 359.83139,z -0.941925526,a 87.5949631,b 2.26507401,c -93.213501,s 2,t 43,e1 0.0,e2 0.0,e3 0.0,e4 0.0,e5 0.0,e6 0.0}
DECL FDAT FSWP_60_7112={TOOL_NO 3,BASE_NO 3,IPO_FRAME #BASE}
DECL LDAT LCPDAT25={VEL 2.0,ACC 100.0,APO_DIST 100.0,APO_FAC 50.0}
DECL E6POS XSWP_60_7114={x 189.108398,y 385.609589,z -1.62237799,a 87.5948792,b 2.26407909,c -93.2117233,s 2,t 43,e1 0.0,e2 0.0,e3 0.0,e4 0.0,e5 0.0,e6 0.0}
DECL FDAT FSWP_60_7114={TOOL_NO 3,BASE_NO 3,IPO_FRAME #BASE}
DECL LDAT LCPDAT26={VEL 2.0,ACC 100.0,APO_DIST 100.0,APO_FAC 50.0}
DECL E6POS XSWP_60_7028={x 186.637604,y 359.650604,z -2.82670903,a 87.5952301,b 2.26461196,c -93.2133102,s 2,t 43,e1 0.0,e2 0.0,e3 0.0,e4 0.0,e5 0.0,e6 0.0}
DECL FDAT FSWP_60_7028={TOOL_NO 3,BASE_NO 3,IPO_FRAME #BASE}
DECL E6POS XSWP_60_7116={x 189.681702,y 419.289215,z 33.1552887,a 87.7462769,b -1.24117994,c -92.174263,s 2,t 43,e1 0.0,e2 0.0,e3 0.0,e4 0.0,e5 0.0,e6 0.0}
DECL FDAT FSWP_60_7116={TOOL_NO 3,BASE_NO 3,IPO_FRAME #BASE}
DECL LDAT LCPDAT27={VEL 2.0,ACC 100.0,APO_DIST 100.0,APO_FAC 50.0}
DECL E6POS XSWP_60_7118={x 181.490906,y 418.84259,z 53.1533203,a 87.8234634,b -5.40211916,c -93.2266388,s 2,t 43,e1 0.0,e2 0.0,e3 0.0,e4 0.0,e5 0.0,e6 0.0}
DECL FDAT FSWP_60_7118={TOOL_NO 3,BASE_NO 3,IPO_FRAME #BASE}
DECL LDAT LCPDAT28={VEL 2.0,ACC 100.0,APO_DIST 100.0,APO_FAC 50.0}
DECL E6POS XSWP_60_7120={x 189.297699,y 423.653015,z 78.365387,a 87.8189468,b -5.40071011,c -93.2256775,s 2,t 43,e1 0.0,e2 0.0,e3 0.0,e4 0.0,e5 0.0,e6 0.0}
DECL FDAT FSWP_60_7120={TOOL_NO 3,BASE_NO 3,IPO_FRAME #BASE}
DECL LDAT LCPDAT29={VEL 2.0,ACC 100.0,APO_DIST 100.0,APO_FAC 50.0}
DECL E6POS XSWP_60_7121={x 181.620407,y 347.470306,z 83.9234619,a 87.8192062,b -5.4038291,c -93.2219467,s 2,t 43,e1 0.0,e2 0.0,e3 0.0,e4 0.0,e5 0.0,e6 0.0}
DECL FDAT FSWP_60_7121={TOOL_NO 3,BASE_NO 3,IPO_FRAME #BASE}
DECL PDAT PPDAT33={VEL 100.0,ACC 80.0,APO_DIST 100.0}
DECL E6POS XSWP_60_7122={x 181.620407,y 347.470306,z 83.9234619,a 87.8192062,b -5.4038291,c -93.2219467,s 2,t 43,e1 0.0,e2 0.0,e3 0.0,e4 0.0,e5 0.0,e6 0.0}
DECL FDAT FSWP_60_7122={TOOL_NO 3,BASE_NO 3,IPO_FRAME #BASE}
DECL PDAT PPDAT34={VEL 100.0,ACC 80.0,APO_DIST 100.0}
DECL E6POS XSWP_60_7123={x -147.606903,y 344.160706,z 83.5968781,a 87.8187332,b -5.40472984,c -93.2222366,s 2,t 42,e1 0.0,e2 0.0,e3 0.0,e4 0.0,e5 0.0,e6 0.0}
DECL FDAT FSWP_60_7123={TOOL_NO 3,BASE_NO 3,IPO_FRAME #BASE}
DECL PDAT PPDAT35={VEL 100.0,ACC 80.0,APO_DIST 100.0}
DECL E6POS XSWP_60_7124={x -373.179199,y 990.898926,z -71.8238373,a 96.4663162,b 6.40630579,c -88.1937637,s 2,t 42,e1 0.0,e2 0.0,e3 0.0,e4 0.0,e5 0.0,e6 0.0}
DECL FDAT FSWP_60_7124={TOOL_NO 3,BASE_NO 3,IPO_FRAME #BASE}
DECL PDAT PPDAT36={VEL 100.0,ACC 80.0,APO_DIST 100.0}
DECL E6POS XSWP_60_7125={x -938.606628,y 703.750183,z 612.628296,a 165.017105,b 23.1202908,c 13.1029396,s 2,t 42,e1 0.0,e2 0.0,e3 0.0,e4 0.0,e5 0.0,e6 0.0}
DECL FDAT FSWP_60_7125={TOOL_NO 3,BASE_NO 3,IPO_FRAME #BASE}
DECL PDAT PPDAT37={VEL 100.0,ACC 80.0,APO_DIST 100.0}
DECL E6POS XSWP_60_7126={x -936.03772,y 1095.39502,z 612.167786,a 165.015793,b 23.1197605,c 13.09867,s 2,t 43,e1 0.0,e2 0.0,e3 0.0,e4 0.0,e5 0.0,e6 0.0}
DECL FDAT FSWP_60_7126={TOOL_NO 3,BASE_NO 3,IPO_FRAME #BASE}
DECL PDAT PPDAT38={VEL 100.0,ACC 80.0,APO_DIST 100.0}
DECL E6POS XSWP_60_7234={x 205.6577,y 368.187012,z 389.243713,a -89.9944229,b 62.69561,c 90.0030975,s 2,t 43,e1 0.0,e2 0.0,e3 0.0,e4 0.0,e5 0.0,e6 0.0}
DECL FDAT FSWP_60_7234={TOOL_NO 3,BASE_NO 3,IPO_FRAME #BASE}
DECL E6POS XSWP_60_7228={x 206.997299,y 237.645493,z 384.287994,a -90.0011597,b 62.6945915,c 89.9988098,s 2,t 43,e1 0.0,e2 0.0,e3 0.0,e4 0.0,e5 0.0,e6 0.0}
DECL FDAT FSWP_60_7228={TOOL_NO 3,BASE_NO 3,IPO_FRAME #BASE}
DECL E6POS XSWP_60_7226={x 207.525299,y 187.710403,z 383.361206,a -90.0016327,b 62.6922607,c 89.9979324,s 2,t 43,e1 0.0,e2 0.0,e3 0.0,e4 0.0,e5 0.0,e6 0.0}
DECL FDAT FSWP_60_7226={TOOL_NO 3,BASE_NO 3,IPO_FRAME #BASE}
DECL E6POS XSWP_60_7224={x 206.951508,y 141.325897,z 384.747589,a -89.9992218,b 54.2501106,c 89.9959335,s 2,t 43,e1 0.0,e2 0.0,e3 0.0,e4 0.0,e5 0.0,e6 0.0}
DECL FDAT FSWP_60_7224={TOOL_NO 3,BASE_NO 3,IPO_FRAME #BASE}
DECL E6POS XSWP_60_7250={x 180.742096,y 249.745895,z 487.002686,a -73.5239868,b 45.4169807,c 112.489998,s 2,t 11,e1 0.0,e2 0.0,e3 0.0,e4 0.0,e5 0.0,e6 0.0}
DECL FDAT FSWP_60_7250={TOOL_NO 3,BASE_NO 3,IPO_FRAME #BASE}
DECL E6POS XSWP_60_9324={x 213.778198,y 837.778687,z 419.142395,a -89.9829102,b 86.8916779,c 90.0147095,s 2,t 43,e1 0.0,e2 0.0,e3 0.0,e4 0.0,e5 0.0,e6 0.0}
DECL FDAT FSWP_60_9324={TOOL_NO 3,BASE_NO 3,IPO_FRAME #BASE}
DECL E6POS XSWP_60_9326={x 213.139099,y 813.078918,z 427.233307,a -90.0939331,b 86.8945618,c 89.9068604,s 2,t 43,e1 0.0,e2 0.0,e3 0.0,e4 0.0,e5 0.0,e6 0.0}
DECL FDAT FSWP_60_9326={TOOL_NO 3,BASE_NO 3,IPO_FRAME #BASE}
DECL E6POS XSWP_60_9328={x 212.856506,y 785.223877,z 444.833801,a -90.077713,b 86.8955765,c 89.9235229,s 2,t 43,e1 0.0,e2 0.0,e3 0.0,e4 0.0,e5 0.0,e6 0.0}
DECL FDAT FSWP_60_9328={TOOL_NO 3,BASE_NO 3,IPO_FRAME #BASE}
DECL E6POS XSWP_60_9330={x 212.668396,y 756.48938,z 464.045013,a -90.0296097,b 86.8944778,c 89.9698868,s 2,t 43,e1 0.0,e2 0.0,e3 0.0,e4 0.0,e5 0.0,e6 0.0}
DECL FDAT FSWP_60_9330={TOOL_NO 3,BASE_NO 3,IPO_FRAME #BASE}
DECL E6POS XSWP_60_9332={x 213.027802,y 725.344971,z 473.002106,a 90.0005112,b 70.9205475,c -89.9997635,s 2,t 43,e1 0.0,e2 0.0,e3 0.0,e4 0.0,e5 0.0,e6 0.0}
DECL FDAT FSWP_60_9332={TOOL_NO 3,BASE_NO 3,IPO_FRAME #BASE}
DECL E6POS XSWP_60_9334={x 212.014206,y 692.942383,z 474.529114,a -90.0135422,b 86.1573029,c 89.9863434,s 2,t 43,e1 0.0,e2 0.0,e3 0.0,e4 0.0,e5 0.0,e6 0.0}
DECL FDAT FSWP_60_9334={TOOL_NO 3,BASE_NO 3,IPO_FRAME #BASE}
DECL E6POS XSWP_60_9336={x 211.981094,y 660.391724,z 475.128998,a -89.9976578,b 56.1076393,c 90.0009232,s 2,t 43,e1 0.0,e2 0.0,e3 0.0,e4 0.0,e5 0.0,e6 0.0}
DECL FDAT FSWP_60_9336={TOOL_NO 3,BASE_NO 3,IPO_FRAME #BASE}
DECL E6POS XSWP_60_9338={x 211.712708,y 634.351624,z 473.975708,a -90.0018463,b 58.2456512,c 89.9996338,s 2,t 43,e1 0.0,e2 0.0,e3 0.0,e4 0.0,e5 0.0,e6 0.0}
DECL FDAT FSWP_60_9338={TOOL_NO 3,BASE_NO 3,IPO_FRAME #BASE}
DECL E6POS XSWP_60_9340={x 211.288498,y 608.372925,z 473.977295,a -90.0021973,b 59.0436783,c 89.997879,s 2,t 43,e1 0.0,e2 0.0,e3 0.0,e4 0.0,e5 0.0,e6 0.0}
DECL FDAT FSWP_60_9340={TOOL_NO 3,BASE_NO 3,IPO_FRAME #BASE}
DECL E6POS XSWP_60_9342={x 211.976898,y 582.396973,z 475.673798,a -90.0029907,b 59.7204399,c 89.9963303,s 2,t 43,e1 0.0,e2 0.0,e3 0.0,e4 0.0,e5 0.0,e6 0.0}
DECL FDAT FSWP_60_9342={TOOL_NO 3,BASE_NO 3,IPO_FRAME #BASE}
DECL E6POS XSWP_60_9344={x 212.347397,y 556.409424,z 475.394012,a -90.0009232,b 60.0734215,c 89.9982071,s 2,t 43,e1 0.0,e2 0.0,e3 0.0,e4 0.0,e5 0.0,e6 0.0}
DECL FDAT FSWP_60_9344={TOOL_NO 3,BASE_NO 3,IPO_FRAME #BASE}
DECL E6POS XSWP_60_9214={x 211.360001,y 441.117401,z 482.715515,a -89.9957428,b 60.0033989,c 90.0009232,s 2,t 43,e1 0.0,e2 0.0,e3 0.0,e4 0.0,e5 0.0,e6 0.0}
DECL FDAT FSWP_60_9214={TOOL_NO 3,BASE_NO 3,IPO_FRAME #BASE}
DECL E6POS XSWP_60_9210={x 212.619003,y 431.033905,z 441.063385,a -89.9974365,b 61.5314484,c 90.0030136,s 2,t 43,e1 0.0,e2 0.0,e3 0.0,e4 0.0,e5 0.0,e6 0.0}
DECL FDAT FSWP_60_9210={TOOL_NO 3,BASE_NO 3,IPO_FRAME #BASE}
DECL E6POS XSWP_60_9208={x 213.415604,y 416.660614,z 400.161407,a -90.01297,b 62.6892014,c 89.9869919,s 2,t 43,e1 0.0,e2 0.0,e3 0.0,e4 0.0,e5 0.0,e6 0.0}
DECL FDAT FSWP_60_9208={TOOL_NO 3,BASE_NO 3,IPO_FRAME #BASE}
DECL E6POS XSWP_60_9218={x 213.644608,y 88.2997208,z 381.914398,a -89.993103,b 44.4734001,c 89.9886169,s 2,t 43,e1 0.0,e2 0.0,e3 0.0,e4 0.0,e5 0.0,e6 0.0}
DECL FDAT FSWP_60_9218={TOOL_NO 3,BASE_NO 3,IPO_FRAME #BASE}
DECL E6POS XSWP_60_9216={x 214.267807,y 40.2348785,z 382.988708,a -89.9609222,b 44.4720802,c 89.994957,s 2,t 43,e1 0.0,e2 0.0,e3 0.0,e4 0.0,e5 0.0,e6 0.0}
DECL FDAT FSWP_60_9216={TOOL_NO 3,BASE_NO 3,IPO_FRAME #BASE}
DECL E6POS XSWP_60_9257={x 187.022995,y 0.48173669,z 486.798096,a -80.9865265,b 30.2971096,c 107.446701,s 2,t 11,e1 0.0,e2 0.0,e3 0.0,e4 0.0,e5 0.0,e6 0.0}
DECL FDAT FSWP_60_9257={TOOL_NO 3,BASE_NO 3,IPO_FRAME #BASE}
DECL E6POS XSWP_60_9256={x 185.367905,y 50.2967796,z 488.660004,a -80.3128967,b 32.1276207,c 107.792999,s 2,t 11,e1 0.0,e2 0.0,e3 0.0,e4 0.0,e5 0.0,e6 0.0}
DECL FDAT FSWP_60_9256={TOOL_NO 3,BASE_NO 3,IPO_FRAME #BASE}
DECL E6POS XSWP_60_9254={x 184.982697,y 92.7076263,z 488.997986,a -80.3136063,b 32.1282005,c 107.791496,s 2,t 11,e1 0.0,e2 0.0,e3 0.0,e4 0.0,e5 0.0,e6 0.0}
DECL FDAT FSWP_60_9254={TOOL_NO 3,BASE_NO 3,IPO_FRAME #BASE}
DECL E6POS XSWP_60_9234={x 206.436905,y 388.897705,z 414.245209,a -43.1899681,b 69.0715408,c 138.711807,s 2,t 43,e1 0.0,e2 0.0,e3 0.0,e4 0.0,e5 0.0,e6 0.0}
DECL FDAT FSWP_60_9234={TOOL_NO 3,BASE_NO 3,IPO_FRAME #BASE}
DECL LDAT LCPDAT30={VEL 2.0,ACC 100.0,APO_DIST 100.0,APO_FAC 50.0}
ENDDAT
